// TIA Portal V17 export
// export: Created 2023-02-13T11:16:04.1669304Z, ExportSetting WithDefaults, DisplayName Totally Integrated Automation Portal, DisplayVersion V17, DisplayName TIA Portal Openness, DisplayVersion V17, DisplayName TIA Portal Teamcenter Gateway, DisplayVersion V17, DisplayName TIA Portal Version Control Interface, DisplayVersion V17, DisplayName SINAMICS Startdrive Advanced, DisplayVersion V17, DisplayName SINAMICS Startdrive G130, G150, S120, S150, SINAMICS MV, S210, DisplayVersion V17, DisplayName SINAMICS Startdrive G110M, G120, G120C, G120D, G120P, G115D, DisplayVersion V17, DisplayName STEP 7 Professional, DisplayVersion V17, DisplayName STEP 7 Safety, DisplayVersion V17, DisplayName WinCC Professional, DisplayVersion V17
DATA_BLOCK "Preparation to Blend"   // DB462
{ S7_Optimized_Access := 'FALSE' }
VERSION : 0.1
// stored: AutoNumber false, DBAccessibleFromOPCUA true, DBAccessibleFromWebserver true, IsOnlyStoredInLoadMemory false, IsWriteProtectedInAS false
   VAR
      "T-51_HW" : Struct
         Tank_Available : Bool;
         Valve_Open : Bool;
         Pump_Run : Bool;
         Product_Ready : Bool;
         freeBool_5 : Bool;
         Level : Bool;
         freeReal_2 : Bool;
         freeReal_3 : Bool;
         freeReal_4 : Bool;
         freeReal_5 : Bool;
      END_STRUCT;
      "T-02_ChiliAwetan_1" : Struct
         Tank_Available : Bool;
         Valve_Open : Bool;
         Pump_Run : Bool;
         Product_Ready : Bool;
         freeBool_5 : Bool;
         Level : Real;
         freeReal_2 : Real;
         freeReal_3 : Real;
         freeReal_4 : Real;
         freeReal_5 : Real;
      END_STRUCT;
      "T-03_ChiliAwetan_2" : Struct
         Tank_Available : Bool;
         Valve_Open : Bool;
         Pump_Run : Bool;
         Product_Ready : Bool;
         freeBool_5 : Bool;
         Level : Real;
         freeReal_2 : Real;
         freeReal_3 : Real;
         freeReal_4 : Real;
         freeReal_5 : Real;
      END_STRUCT;
      "T-04_ChiliAwetan_3" : Struct
         Tank_Available : Bool;
         Valve_Open : Bool;
         Pump_Run : Bool;
         Product_Ready : Bool;
         freeBool_5 : Bool;
         Level : Real;
         freeReal_2 : Real;
         freeReal_3 : Real;
         freeReal_4 : Real;
         freeReal_5 : Real;
      END_STRUCT;
      "T-05_Tomato" : Struct
         Tank_Available : Bool;
         Valve_Open : Bool;
         Pump_Run : Bool;
         Product_Ready : Bool;
         freeBool_5 : Bool;
         Level : Real;
         freeReal_2 : Real;
         freeReal_3 : Real;
         freeReal_4 : Real;
         freeReal_5 : Real;
      END_STRUCT;
      "T-06_ChiliFresh_1" : Struct
         Tank_Available : Bool;
         Valve_Open : Bool;
         Pump_Run : Bool;
         Product_Ready : Bool;
         freeBool_5 : Bool;
         Level : Real;
         freeReal_2 : Real;
         freeReal_3 : Real;
         freeReal_4 : Real;
         freeReal_5 : Real;
      END_STRUCT;
      "T-07_ChiliFresh_2" : Struct
         Tank_Available : Bool;
         Valve_Open : Bool;
         Pump_Run : Bool;
         Product_Ready : Bool;
         freeBool_5 : Bool;
         Level : Real;
         freeReal_2 : Real;
         freeReal_3 : Real;
         freeReal_4 : Real;
         freeReal_5 : Real;
      END_STRUCT;
      "T-08_ChiliFresh_3" : Struct
         Tank_Available : Bool;
         Valve_Open : Bool;
         Pump_Run : Bool;
         Product_Ready : Bool;
         freeBool_5 : Bool;
         Level : Real;
         freeReal_2 : Real;
         freeReal_3 : Real;
         freeReal_4 : Real;
         freeReal_5 : Real;
      END_STRUCT;
      "T-09_Garlic" : Struct
         Tank_Available : Bool;
         Valve_Open : Bool;
         Pump_Run : Bool;
         Product_Ready : Bool;
         freeBool_5 : Bool;
         Level : Real;
         freeReal_2 : Real;
         freeReal_3 : Real;
         freeReal_4 : Real;
         freeReal_5 : Real;
      END_STRUCT;
      "T-10_Vinegar" : Struct
         Tank_Available : Bool;
         Valve_Open : Bool;
         Pump_Run : Bool;
         Product_Ready : Bool;
         freeBool_5 : Bool;
         Level : Real;
         freeReal_2 : Real;
         freeReal_3 : Real;
         freeReal_4 : Real;
         freeReal_5 : Real;
      END_STRUCT;
      Header_1_CIP : Bool;
      Header_2_CIP : Bool;
      Header_1_Flushing : Bool;
      Header_2_Flushing : Bool;
      freeBool_5 : Bool;
      freeBool_6 : Bool;
      freeBool_7 : Bool;
      freeBool_8 : Bool;
      freeBool_9 : Bool;
      freeBool_10 : Bool;
      freeBool_11 : Bool;
      freeBool_12 : Bool;
      freeBool_13 : Bool;
      freeBool_14 : Bool;
      freeBool_15 : Bool;
      freeBool_16 : Bool;
      freeReal_1 : Real;
      freeReal_2 : Real;
      freeReal_3 : Real;
      freeReal_4 : Real;
      freeReal_5 : Real;
      freeReal_6 : Real;
      freeReal_7 : Real;
      freeReal_8 : Real;
      freeReal_9 : Real;
      freeReal_10 : Real;
      freeReal_11 : Real;
      freeReal_12 : Real;
      freeReal_13 : Real;
      freeReal_14 : Real;
      freeReal_15 : Real;
   END_VAR
BEGIN
END_DATA_BLOCK
